{attribute addProperty BoxType "EL3632-0000-0022"}
{attribute addProperty Id "UnderrangeBIT10.1251OverrangeBIT10.1252Limit_1_BIT_0BIT10.1253Limit_1_BIT_1BIT10.1253Limit_2_BIT_0BIT10.1255Limit_2_BIT_1BIT10.1255ErrorBIT10.1257Sync_errorBIT10.12514TxPDO_StateBIT10.12515TxPDO_ToggleBIT10.12516"}
{attribute addProperty CRC "2219972760"}
{attribute addProperty SizeInBites "16"}
{attribute addProperty SizeInBytes "2"}
TYPE STATUS_84521898 :
STRUCT
	{attribute addProperty Name "Underrange"}
	Underrange : BIT;
	{attribute addProperty Name "Overrange"}
	Overrange : BIT;
	{attribute addProperty Name "Limit_1"}
	Limit_1_BIT_0 : BIT;
	{attribute addProperty Name "Limit_1"}
	Limit_1_BIT_1 : BIT;
	{attribute addProperty Name "Limit_2"}
	Limit_2_BIT_0 : BIT;
	{attribute addProperty Name "Limit_2"}
	Limit_2_BIT_1 : BIT;
	{attribute addProperty Name "Error"}
	Error : BIT;
	{attribute 'hide'}
	reserve_1_BIT_0 : BIT;
	{attribute 'hide'}
	reserve_1_BIT_1 : BIT;
	{attribute 'hide'}
	reserve_1_BIT_2 : BIT;
	{attribute 'hide'}
	reserve_1_BIT_3 : BIT;
	{attribute 'hide'}
	reserve_1_BIT_4 : BIT;
	{attribute 'hide'}
	reserve_1_BIT_5 : BIT;
	{attribute addProperty Name "Sync_error"}
	Sync_error : BIT;
	{attribute addProperty Name "TxPDO_State"}
	TxPDO_State : BIT;
	{attribute addProperty Name "TxPDO_Toggle"}
	TxPDO_Toggle : BIT;
END_STRUCT
END_TYPE

(* stored: Version 1.2.0.0, ProductVersion 3.1.4024.9
   DUT STATUS_84521898: Id {cdc12883-3907-4fe0-80fd-8ae61df5b2e2} *)
